FUNCTION FindMinMax 
VAR_INPUT
	aWeight : ARRAY[1..20] OF REAL;
END_VAR
VAR_IN_OUT
    minWeight : REAL;
	maxWeight : REAL;
END_VAR
VAR
	i : INT;
	bFirst   : BOOL := TRUE;
END_VAR

FOR i := 1 TO 20 DO

    IF (aWeight[i] >= 50.0) AND (aWeight[i] <= 500.0) THEN
        
        IF bFirst THEN
            minWeight := aWeight[i];
            maxWeight := aWeight[i];
            bFirst := FALSE;
        ELSE
            
            IF aWeight[i] > maxWeight THEN
                maxWeight := aWeight[i];
            END_IF
            
            IF aWeight[i] < minWeight THEN
                minWeight := aWeight[i];
            END_IF
            
        END_IF
        
    END_IF

END_FOR


IF bFirst THEN
    minWeight := 0.0;
    maxWeight := 0.0;
END_IF

END_FUNCTION

(* stored: Version 1.1.0.1, ProductVersion 3.1.4024.16
   POU FindMinMax: Id {d8c3f14f-a8ff-4548-a67d-a8a902cf1ffe}, SpecialFunc None *)
